Yaskawa INFORM job: PICK.JBI

/JOB
//NAME PICK-DAR
//POS
///NPOS 0,0,0,1,0,0
///TOOL 0
///POSTYPE ROBOT
///RECTAN
///RCONF 0,0,0,0,0,0,0,0,0,0,0,0,0,0,0,0,0,0,0,0,0,0,0,0
P00003=237.030,36.158,-47.377,-179.9824,-0.0082,0.0088
//INST
///DATE 2019/05/19 12:33
///ATTR SC,RW
///GROUP1 RB1
NOP
*PICK
MOVL P003 V=187.0
IFTHENEXP B003=1 OREXP B006=1 OREXP B007=1
	 DOUT OT#(1) ON
	 RET
ENDIF
JUMP *PICK
END
